(* CODESYS project HFX_research_EMMS_.project

Project tree, tasks and I/O mapping:
  Device : CR1201, ifm electronic, order no. PDM360NG, version 3.3.0.2
    application Application
      libraries: Standard, * (System); VisuDialogs, * (System); CAA CiA 405, 3.5.8.0 (CAA Technical Workgroup)
      task MainTask (cyclic, interval t#20ms, priority 1) calls PLC_PRG
      task VISU_TASK (cyclic, interval t#20ms, priority 15) calls VisuElems.Visu_Prg
      task TrendRecordingTask (cyclic, interval 100 ms, priority 31) calls VisuTrendStorageAccess.GlobalInstances.g_TrendRecordingManager.CyclicCall
      program PLC_PRG [ST]
      visualisation Main_sys
      visualisation Battery_sys
      visualisation Hydrogen_Fuel_cell_sys
      visualisation Main_Overview
      visualisation Hydrogen_Tanks
      visualisation Machine_system_properties
      visualisation Control_System_Simulation
      visualisation Visualization
      visualisation electric_motor
      visualisation Hydraulic_System
      visualisation Cooling_system
      visualisation camera_system
      image pool ImagePool
    System_Info : System_Info, ifm electronic, version 3.3.0.2
    Local_IO : Local IO, ifm electronic, version 3.3.0.2
      Inputs : Inputs, ifm electronic, version 3.3.0.2
          input  IN0000 : IN_MULTIFUNCTION_B_INPUT_MAPPING_TYPE  // IN0000
      Outputs : Outputs, ifm electronic, version 3.3.0.2
          output OUT0000 : OUT_DIGITAL_A_OUTPUT_MAPPING_TYPE  // OUT0000
      System_Inputs : System_Inputs, ifm electronic, version 3.3.0.2
          input  uiVoltageVBB30 : UINT  // Voltage VBB30
          input  uiVoltageVBB15 : UINT  // Voltage VBB15
          input  iTemperature0 : INT  // Board Temperature 0
          input  iTemperature1 : INT  // Board Temperature 1
          input  uiLightSensor : UINT  // Light Sensor
    HMI : HMI, ifm electronic, version 3.3.0.2
      User_LEDs : User_LEDs, ifm electronic, version 3.3.0.2
          output LED0 : LED_IEC_A_OUTPUT_MAPPING_TYPE  // User LED 0
      LCD_Backlight : LCD Backlight, ifm electronic, version 3.3.0.2
          output uiBacklightBrightness AT %QW5 : UINT  // Brightness
      Buzzer : Buzzer, ifm electronic, version 3.3.0.2
          output uiBuzzerFreq : UINT  // Frequency
          output xBuzzerON : BIT  // Buzzer ON
      KeyBoards : KeyBoards, ifm electronic, version 3.3.0.2
        Key_Backlight_settings : Key Backlight settings, ifm electronic, version 3.3.0.2
            output xNightModeON AT %QX14.1 : BIT  // Night Mode ON
        Key_Mapping : Key Mapping, ifm electronic, version 3.3.0.2
        Keys : Keys, ifm electronic, version 3.3.0.2
          LEDs_Keyboard_1 : LEDs Keyboard 1, ifm electronic, version 3.3.0.2
              output LEDsKeyboard1 AT %QW8 : WORD  // LEDsKeyboard1
          LEDs_Keyboard_3 : LEDs Keyboard 3, ifm electronic, version 3.3.0.2
              output LEDsKeyboard3 AT %QW9 : WORD  // LEDs Keyboard 3
    Communication : Communication, ifm electronic, version 3.3.0.2
      Ethernet : Ethernet, ifm electronic, version 3.3.0.2
      CAN : CAN, ifm electronic, version 3.3.0.2
        CANbus : CANbus, ifm electronic, version 1.0.0.0
            settings: Baudrate = 125; NetID = 1
          CANopen_Manager : CANopen_Manager, 3S - Smart Software Solutions GmbH, version 3.5.7.20
              settings: ConfigVersion = 50659584
            JN2100 : JN2100, ifm electornic GmbH, order no. JN2100, version Revision=16#000000AA, FileVersion=1.1, File=inclinationsensor_JNJN2100_V2.5.4.eds
                settings: General Options.Create all SDOs = TRUE; NODEIDSAVED = 10; SDO Timeout = 1000000; Explicit Deactivate PDOs = TRUE; PDO_Autoconfig = FALSE; EXPERTSETTINGS = True; Emergency-General Parameters.Emergency COBID = 16#0000008A; Heartbeat-Producer Time = 200; PDO 16#1800.COBID = 16#0000018A; PDO 16#1800.Transmission Type = 16#FE; Process by CANopenManager = TRUE; PDO 16#1801.COBID = 16#0000028A; PDO 16#1801.Transmission Type = 16#FE; Process by CANopenManager = TRUE; PDO 16#1802.COBID = 16#0000038A; PDO 16#1802.Transmission Type = 16#FE; Process by CANopenManager = TRUE; PDO 16#1803.COBID = 16#0000048A; PDO 16#1803.Transmission Type = 16#FE; Process by CANopenManager = TRUE; Slope long16.Subindex = 16#00; Slope lateral16.Subindex = 16#00; Slope long32.Subindex = 16#00; Slope lateral32.Subindex = 16#00; v effektive vector magnitude.Subindex = 16#00; a peak vector magnitude.Subindex = 16#00; a x vector.Subindex = 16#00; a y vector.Subindex = 16#00; a z vector.Subindex = 16#00; SDO List.Set Guardtime.Index = 16#100C; SDO List.Set Guardtime.Subindex = 16#00; SDO List.Set Guardtime.Value = 16#00000000; SDO List.Set Guardtime.Size = 16; SDO List.Set Guardtime.AbortIfError = FALSE; SDO List.Set Guardtime.JumpToLine = FALSE; SDO List.Set Guardtime.Line = 0; SDO List.Set Lifetime.Index = 16#100D; SDO List.Set Lifetime.Subindex = 16#00; SDO List.Set Lifetime.Value = 16#00000000; SDO List.Set Lifetime.Size = 8;
                  SDO List.Set Lifetime.AbortIfError = FALSE; SDO List.Set Lifetime.JumpToLine = FALSE; SDO List.Set Lifetime.Line = 0; SDO List.Set Heartbeat Producer.Index = 16#1017; SDO List.Set Heartbeat Producer.Subindex = 16#00; SDO List.Set Heartbeat Producer.Value = 16#000000C8; SDO List.Set Heartbeat Producer.Size = 16; SDO List.Set Heartbeat Producer.AbortIfError = FALSE; SDO List.Set Heartbeat Producer.JumpToLine = FALSE; SDO List.Set Heartbeat Producer.Line = 0; SDO List.Disable PDO.Index = 16#1800; SDO List.Disable PDO.Subindex = 16#01; SDO List.Disable PDO.Value = 16#8000018A; SDO List.Disable PDO.Size = 32; SDO List.Disable PDO.AbortIfError = FALSE; SDO List.Disable PDO.JumpToLine = FALSE; SDO List.Disable PDO.Line = 0; SDO List.Set transmission type.Index = 16#1800; SDO List.Set transmission type.Subindex = 16#02; SDO List.Set transmission type.Value = 16#FE; SDO List.Set transmission type.Size = 8; SDO List.Set transmission type.AbortIfError = FALSE; SDO List.Set transmission type.JumpToLine = FALSE; SDO List.Set transmission type.Line = 0; SDO List.Set inhibit time.Index = 16#1800; SDO List.Set inhibit time.Subindex = 16#03; SDO List.Set inhibit time.Value = 16#0000; SDO List.Set inhibit time.Size = 16; SDO List.Set inhibit time.AbortIfError = FALSE; SDO List.Set inhibit time.JumpToLine = FALSE; SDO List.Set inhibit time.Line = 0; SDO List.Set event time.Index = 16#1800; SDO List.Set event time.Subindex = 16#05; SDO List.Set event time.Value = 16#000A; SDO List.Set event time.Size = 16; SDO List.Set event time.AbortIfError = FALSE; SDO List.Set event time.JumpToLine = FALSE; SDO List.Set event time.Line = 0; SDO List.Clear pdo mapping.Index = 16#1A00; SDO List.Clear pdo mapping.Subindex = 16#00;
                  SDO List.Clear pdo mapping.Value = 16#0; SDO List.Clear pdo mapping.Size = 8; SDO List.Clear pdo mapping.AbortIfError = FALSE; SDO List.Clear pdo mapping.JumpToLine = FALSE; SDO List.Clear pdo mapping.Line = 0; SDO List.Set Mapping.Index = 16#1A00; SDO List.Set Mapping.Subindex = 16#01; SDO List.Set Mapping.Value = 16#60100010; SDO List.Set Mapping.Size = 32; SDO List.Set Mapping.AbortIfError = FALSE; SDO List.Set Mapping.JumpToLine = FALSE; SDO List.Set Mapping.Line = 0; SDO List.Set Mapping.Index = 16#1A00; SDO List.Set Mapping.Subindex = 16#02; SDO List.Set Mapping.Value = 16#60200010; SDO List.Set Mapping.Size = 32; SDO List.Set Mapping.AbortIfError = FALSE; SDO List.Set Mapping.JumpToLine = FALSE; SDO List.Set Mapping.Line = 0; SDO List.Set number of mappings.Index = 16#1A00; SDO List.Set number of mappings.Subindex = 16#00; SDO List.Set number of mappings.Value = 16#02; SDO List.Set number of mappings.Size = 8; SDO List.Set number of mappings.AbortIfError = FALSE; SDO List.Set number of mappings.JumpToLine = FALSE; SDO List.Set number of mappings.Line = 0; SDO List.Set and enable COB-ID.Index = 16#1800; SDO List.Set and enable COB-ID.Subindex = 16#01; SDO List.Set and enable COB-ID.Value = 16#0000018A; SDO List.Set and enable COB-ID.Size = 32; SDO List.Set and enable COB-ID.AbortIfError = FALSE; SDO List.Set and enable COB-ID.JumpToLine = FALSE; SDO List.Set and enable COB-ID.Line = 0; SDO List.Disable PDO.Index = 16#1801; SDO List.Disable PDO.Subindex = 16#01; SDO List.Disable PDO.Value = 16#8000028A; SDO List.Disable PDO.Size = 32; SDO List.Disable PDO.AbortIfError = FALSE; SDO List.Disable PDO.JumpToLine = FALSE; SDO List.Disable PDO.Line = 0;
                  SDO List.Set transmission type.Index = 16#1801; SDO List.Set transmission type.Subindex = 16#02; SDO List.Set transmission type.Value = 16#FE; SDO List.Set transmission type.Size = 8; SDO List.Set transmission type.AbortIfError = FALSE; SDO List.Set transmission type.JumpToLine = FALSE; SDO List.Set transmission type.Line = 0; SDO List.Set inhibit time.Index = 16#1801; SDO List.Set inhibit time.Subindex = 16#03; SDO List.Set inhibit time.Value = 16#0000; SDO List.Set inhibit time.Size = 16; SDO List.Set inhibit time.AbortIfError = FALSE; SDO List.Set inhibit time.JumpToLine = FALSE; SDO List.Set inhibit time.Line = 0; SDO List.Set event time.Index = 16#1801; SDO List.Set event time.Subindex = 16#05; SDO List.Set event time.Value = 16#000A; SDO List.Set event time.Size = 16; SDO List.Set event time.AbortIfError = FALSE; SDO List.Set event time.JumpToLine = FALSE; SDO List.Set event time.Line = 0; SDO List.Clear pdo mapping.Index = 16#1A01; SDO List.Clear pdo mapping.Subindex = 16#00; SDO List.Clear pdo mapping.Value = 16#0; SDO List.Clear pdo mapping.Size = 8; SDO List.Clear pdo mapping.AbortIfError = FALSE; SDO List.Clear pdo mapping.JumpToLine = FALSE; SDO List.Clear pdo mapping.Line = 0; SDO List.Set Mapping.Index = 16#1A01; SDO List.Set Mapping.Subindex = 16#01; SDO List.Set Mapping.Value = 16#61100020; SDO List.Set Mapping.Size = 32; SDO List.Set Mapping.AbortIfError = FALSE; SDO List.Set Mapping.JumpToLine = FALSE; SDO List.Set Mapping.Line = 0; SDO List.Set Mapping.Index = 16#1A01; SDO List.Set Mapping.Subindex = 16#02; SDO List.Set Mapping.Value = 16#61200020; SDO List.Set Mapping.Size = 32; SDO List.Set Mapping.AbortIfError = FALSE;
                  SDO List.Set Mapping.JumpToLine = FALSE; SDO List.Set Mapping.Line = 0; SDO List.Set number of mappings.Index = 16#1A01; SDO List.Set number of mappings.Subindex = 16#00; SDO List.Set number of mappings.Value = 16#02; SDO List.Set number of mappings.Size = 8; SDO List.Set number of mappings.AbortIfError = FALSE; SDO List.Set number of mappings.JumpToLine = FALSE; SDO List.Set number of mappings.Line = 0; SDO List.Set and enable COB-ID.Index = 16#1801; SDO List.Set and enable COB-ID.Subindex = 16#01; SDO List.Set and enable COB-ID.Value = 16#0000028A; SDO List.Set and enable COB-ID.Size = 32; SDO List.Set and enable COB-ID.AbortIfError = FALSE; SDO List.Set and enable COB-ID.JumpToLine = FALSE; SDO List.Set and enable COB-ID.Line = 0; SDO List.Disable PDO.Index = 16#1802; SDO List.Disable PDO.Subindex = 16#01; SDO List.Disable PDO.Value = 16#8000038A; SDO List.Disable PDO.Size = 32; SDO List.Disable PDO.AbortIfError = FALSE; SDO List.Disable PDO.JumpToLine = FALSE; SDO List.Disable PDO.Line = 0; SDO List.Set transmission type.Index = 16#1802; SDO List.Set transmission type.Subindex = 16#02; SDO List.Set transmission type.Value = 16#FE; SDO List.Set transmission type.Size = 8; SDO List.Set transmission type.AbortIfError = FALSE; SDO List.Set transmission type.JumpToLine = FALSE; SDO List.Set transmission type.Line = 0; SDO List.Set inhibit time.Index = 16#1802; SDO List.Set inhibit time.Subindex = 16#03; SDO List.Set inhibit time.Value = 16#0000; SDO List.Set inhibit time.Size = 16; SDO List.Set inhibit time.AbortIfError = FALSE; SDO List.Set inhibit time.JumpToLine = FALSE; SDO List.Set inhibit time.Line = 0; SDO List.Set event time.Index = 16#1802; SDO List.Set event time.Subindex = 16#05; SDO List.Set event time.Value = 16#000A;
                  SDO List.Set event time.Size = 16; SDO List.Set event time.AbortIfError = FALSE; SDO List.Set event time.JumpToLine = FALSE; SDO List.Set event time.Line = 0; SDO List.Clear pdo mapping.Index = 16#1A02; SDO List.Clear pdo mapping.Subindex = 16#00; SDO List.Clear pdo mapping.Value = 16#0; SDO List.Clear pdo mapping.Size = 8; SDO List.Clear pdo mapping.AbortIfError = FALSE; SDO List.Clear pdo mapping.JumpToLine = FALSE; SDO List.Clear pdo mapping.Line = 0; SDO List.Set Mapping.Index = 16#1A02; SDO List.Set Mapping.Subindex = 16#01; SDO List.Set Mapping.Value = 16#5C100020; SDO List.Set Mapping.Size = 32; SDO List.Set Mapping.AbortIfError = FALSE; SDO List.Set Mapping.JumpToLine = FALSE; SDO List.Set Mapping.Line = 0; SDO List.Set Mapping.Index = 16#1A02; SDO List.Set Mapping.Subindex = 16#02; SDO List.Set Mapping.Value = 16#5C110020; SDO List.Set Mapping.Size = 32; SDO List.Set Mapping.AbortIfError = FALSE; SDO List.Set Mapping.JumpToLine = FALSE; SDO List.Set Mapping.Line = 0; SDO List.Set number of mappings.Index = 16#1A02; SDO List.Set number of mappings.Subindex = 16#00; SDO List.Set number of mappings.Value = 16#02; SDO List.Set number of mappings.Size = 8; SDO List.Set number of mappings.AbortIfError = FALSE; SDO List.Set number of mappings.JumpToLine = FALSE; SDO List.Set number of mappings.Line = 0; SDO List.Set and enable COB-ID.Index = 16#1802; SDO List.Set and enable COB-ID.Subindex = 16#01; SDO List.Set and enable COB-ID.Value = 16#0000038A; SDO List.Set and enable COB-ID.Size = 32; SDO List.Set and enable COB-ID.AbortIfError = FALSE; SDO List.Set and enable COB-ID.JumpToLine = FALSE; SDO List.Set and enable COB-ID.Line = 0; SDO List.Disable PDO.Index = 16#1803;
                  SDO List.Disable PDO.Subindex = 16#01; SDO List.Disable PDO.Value = 16#8000048A; SDO List.Disable PDO.Size = 32; SDO List.Disable PDO.AbortIfError = FALSE; SDO List.Disable PDO.JumpToLine = FALSE; SDO List.Disable PDO.Line = 0; SDO List.Set transmission type.Index = 16#1803; SDO List.Set transmission type.Subindex = 16#02; SDO List.Set transmission type.Value = 16#FE; SDO List.Set transmission type.Size = 8; SDO List.Set transmission type.AbortIfError = FALSE; SDO List.Set transmission type.JumpToLine = FALSE; SDO List.Set transmission type.Line = 0; SDO List.Set inhibit time.Index = 16#1803; SDO List.Set inhibit time.Subindex = 16#03; SDO List.Set inhibit time.Value = 16#0000; SDO List.Set inhibit time.Size = 16; SDO List.Set inhibit time.AbortIfError = FALSE; SDO List.Set inhibit time.JumpToLine = FALSE; SDO List.Set inhibit time.Line = 0; SDO List.Set event time.Index = 16#1803; SDO List.Set event time.Subindex = 16#05; SDO List.Set event time.Value = 16#000A; SDO List.Set event time.Size = 16; SDO List.Set event time.AbortIfError = FALSE; SDO List.Set event time.JumpToLine = FALSE; SDO List.Set event time.Line = 0; SDO List.Clear pdo mapping.Index = 16#1A03; SDO List.Clear pdo mapping.Subindex = 16#00; SDO List.Clear pdo mapping.Value = 16#0; SDO List.Clear pdo mapping.Size = 8; SDO List.Clear pdo mapping.AbortIfError = FALSE; SDO List.Clear pdo mapping.JumpToLine = FALSE; SDO List.Clear pdo mapping.Line = 0; SDO List.Set Mapping.Index = 16#1A03; SDO List.Set Mapping.Subindex = 16#01; SDO List.Set Mapping.Value = 16#5D100010; SDO List.Set Mapping.Size = 32; SDO List.Set Mapping.AbortIfError = FALSE; SDO List.Set Mapping.JumpToLine = FALSE;
                  SDO List.Set Mapping.Line = 0; SDO List.Set Mapping.Index = 16#1A03; SDO List.Set Mapping.Subindex = 16#02; SDO List.Set Mapping.Value = 16#5D110010; SDO List.Set Mapping.Size = 32; SDO List.Set Mapping.AbortIfError = FALSE; SDO List.Set Mapping.JumpToLine = FALSE; SDO List.Set Mapping.Line = 0; SDO List.Set Mapping.Index = 16#1A03; SDO List.Set Mapping.Subindex = 16#03; SDO List.Set Mapping.Value = 16#5D120010; SDO List.Set Mapping.Size = 32; SDO List.Set Mapping.AbortIfError = FALSE; SDO List.Set Mapping.JumpToLine = FALSE; SDO List.Set Mapping.Line = 0; SDO List.Set number of mappings.Index = 16#1A03; SDO List.Set number of mappings.Subindex = 16#00; SDO List.Set number of mappings.Value = 16#03; SDO List.Set number of mappings.Size = 8; SDO List.Set number of mappings.AbortIfError = FALSE; SDO List.Set number of mappings.JumpToLine = FALSE; SDO List.Set number of mappings.Line = 0; SDO List.Set and enable COB-ID.Index = 16#1803; SDO List.Set and enable COB-ID.Subindex = 16#01; SDO List.Set and enable COB-ID.Value = 16#0000048A; SDO List.Set and enable COB-ID.Size = 32; SDO List.Set and enable COB-ID.AbortIfError = FALSE; SDO List.Set and enable COB-ID.JumpToLine = FALSE; SDO List.Set and enable COB-ID.Line = 0; SDO List.Node ID.Index = 16#2000; SDO List.Node ID.Subindex = 16#00; SDO List.Node ID.Value = 10; SDO List.Node ID.Size = 8; SDO List.Node ID.AbortIfError = FALSE; SDO List.Node ID.JumpToLine = FALSE; SDO List.Node ID.Line = 0; SDO List.Baudrate [kbit].Index = 16#2001; SDO List.Baudrate [kbit].Subindex = 16#00; SDO List.Baudrate [kbit].Value = 125; SDO List.Baudrate [kbit].Size = 16;
                  SDO List.Baudrate [kbit].AbortIfError = FALSE; SDO List.Baudrate [kbit].JumpToLine = FALSE; SDO List.Baudrate [kbit].Line = 0; SDO List.Microcontroller Reset.Index = 16#2002; SDO List.Microcontroller Reset.Subindex = 16#00; SDO List.Microcontroller Reset.Value = 0; SDO List.Microcontroller Reset.Size = 8; SDO List.Microcontroller Reset.AbortIfError = FALSE; SDO List.Microcontroller Reset.JumpToLine = FALSE; SDO List.Microcontroller Reset.Line = 0; SDO List.Quadrant Correction.Index = 16#2040; SDO List.Quadrant Correction.Subindex = 16#00; SDO List.Quadrant Correction.Value = 2; SDO List.Quadrant Correction.Size = 8; SDO List.Quadrant Correction.AbortIfError = FALSE; SDO List.Quadrant Correction.JumpToLine = FALSE; SDO List.Quadrant Correction.Line = 0; SDO List.Heater On.Index = 16#2041; SDO List.Heater On.Subindex = 16#00; SDO List.Heater On.Value = 1; SDO List.Heater On.Size = 8; SDO List.Heater On.AbortIfError = FALSE; SDO List.Heater On.JumpToLine = FALSE; SDO List.Heater On.Line = 0; SDO List.Teach Index.Index = 16#2042; SDO List.Teach Index.Subindex = 16#00; SDO List.Teach Index.Value = 2; SDO List.Teach Index.Size = 8; SDO List.Teach Index.AbortIfError = FALSE; SDO List.Teach Index.JumpToLine = FALSE; SDO List.Teach Index.Line = 0; SDO List.FIR Filter Angle.Index = 16#2043; SDO List.FIR Filter Angle.Subindex = 16#00; SDO List.FIR Filter Angle.Value = 2; SDO List.FIR Filter Angle.Size = 8; SDO List.FIR Filter Angle.AbortIfError = FALSE; SDO List.FIR Filter Angle.JumpToLine = FALSE; SDO List.FIR Filter Angle.Line = 0; SDO List.Angle Calculation Algorithm.Index = 16#2044; SDO List.Angle Calculation Algorithm.Subindex = 16#00;
                  SDO List.Angle Calculation Algorithm.Value = 0; SDO List.Angle Calculation Algorithm.Size = 8; SDO List.Angle Calculation Algorithm.AbortIfError = FALSE; SDO List.Angle Calculation Algorithm.JumpToLine = FALSE; SDO List.Angle Calculation Algorithm.Line = 0; SDO List.CAN 120 Ohm Resistor.Index = 16#2045; SDO List.CAN 120 Ohm Resistor.Subindex = 16#00; SDO List.CAN 120 Ohm Resistor.Value = 1; SDO List.CAN 120 Ohm Resistor.Size = 8; SDO List.CAN 120 Ohm Resistor.AbortIfError = FALSE; SDO List.CAN 120 Ohm Resistor.JumpToLine = FALSE; SDO List.CAN 120 Ohm Resistor.Line = 0; SDO List.Zero Index.Index = 16#2046; SDO List.Zero Index.Subindex = 16#00; SDO List.Zero Index.Value = 2; SDO List.Zero Index.Size = 8; SDO List.Zero Index.AbortIfError = FALSE; SDO List.Zero Index.JumpToLine = FALSE; SDO List.Zero Index.Line = 0; SDO List.Measurement Output.Index = 16#2047; SDO List.Measurement Output.Subindex = 16#00; SDO List.Measurement Output.Value = 0; SDO List.Measurement Output.Size = 8; SDO List.Measurement Output.AbortIfError = FALSE; SDO List.Measurement Output.JumpToLine = FALSE; SDO List.Measurement Output.Line = 0; SDO List.Axis Selection v eff - a peak.Index = 16#2048; SDO List.Axis Selection v eff - a peak.Subindex = 16#00; SDO List.Axis Selection v eff - a peak.Value = 7; SDO List.Axis Selection v eff - a peak.Size = 8; SDO List.Axis Selection v eff - a peak.AbortIfError = FALSE; SDO List.Axis Selection v eff - a peak.JumpToLine = FALSE; SDO List.Axis Selection v eff - a peak.Line = 0; SDO List.FIR Filter v eff - a peak.Index = 16#2049; SDO List.FIR Filter v eff - a peak.Subindex = 16#00; SDO List.FIR Filter v eff - a peak.Value = 5; SDO List.FIR Filter v eff - a peak.Size = 8; SDO List.FIR Filter v eff - a peak.AbortIfError = FALSE; SDO List.FIR Filter v eff - a peak.JumpToLine = FALSE; SDO List.FIR Filter v eff - a peak.Line = 0;
                  SDO List.Measurement Range v eff - a peak.Index = 16#204A; SDO List.Measurement Range v eff - a peak.Subindex = 16#00; SDO List.Measurement Range v eff - a peak.Value = 2; SDO List.Measurement Range v eff - a peak.Size = 8; SDO List.Measurement Range v eff - a peak.AbortIfError = FALSE; SDO List.Measurement Range v eff - a peak.JumpToLine = FALSE; SDO List.Measurement Range v eff - a peak.Line = 0; SDO List.Factory Reset.Index = 16#207F; SDO List.Factory Reset.Subindex = 16#00; SDO List.Factory Reset.Value = 0; SDO List.Factory Reset.Size = 8; SDO List.Factory Reset.AbortIfError = FALSE; SDO List.Factory Reset.JumpToLine = FALSE; SDO List.Factory Reset.Line = 0; SDO List.Activate Self Test.Index = 16#4004; SDO List.Activate Self Test.Subindex = 16#01; SDO List.Activate Self Test.Value = 0; SDO List.Activate Self Test.Size = 8; SDO List.Activate Self Test.AbortIfError = FALSE; SDO List.Activate Self Test.JumpToLine = FALSE; SDO List.Activate Self Test.Line = 0; SDO List.Resolution.Index = 16#6000; SDO List.Resolution.Subindex = 16#00; SDO List.Resolution.Value = 100; SDO List.Resolution.Size = 16; SDO List.Resolution.AbortIfError = FALSE; SDO List.Resolution.JumpToLine = FALSE; SDO List.Resolution.Line = 0; SDO List.Slope long16 operating parameter.Index = 16#6011; SDO List.Slope long16 operating parameter.Subindex = 16#00; SDO List.Slope long16 operating parameter.Value = 16#0; SDO List.Slope long16 operating parameter.Size = 8; SDO List.Slope long16 operating parameter.AbortIfError = FALSE; SDO List.Slope long16 operating parameter.JumpToLine = FALSE; SDO List.Slope long16 operating parameter.Line = 0; SDO List.Slope lateral16 operating parameter.Index = 16#6021; SDO List.Slope lateral16 operating parameter.Subindex = 16#00; SDO List.Slope lateral16 operating parameter.Value = 16#0; SDO List.Slope lateral16 operating parameter.Size = 8; SDO List.Slope lateral16 operating parameter.AbortIfError = FALSE;
                  SDO List.Slope lateral16 operating parameter.JumpToLine = FALSE; SDO List.Slope lateral16 operating parameter.Line = 0; SDO List.Slope long32 operating parameter.Index = 16#6111; SDO List.Slope long32 operating parameter.Subindex = 16#00; SDO List.Slope long32 operating parameter.Value = 16#0; SDO List.Slope long32 operating parameter.Size = 8; SDO List.Slope long32 operating parameter.AbortIfError = FALSE; SDO List.Slope long32 operating parameter.JumpToLine = FALSE; SDO List.Slope long32 operating parameter.Line = 0; SDO List.Slope lateral32 operating parameter.Index = 16#6121; SDO List.Slope lateral32 operating parameter.Subindex = 16#00; SDO List.Slope lateral32 operating parameter.Value = 16#0; SDO List.Slope lateral32 operating parameter.Size = 8; SDO List.Slope lateral32 operating parameter.AbortIfError = FALSE; SDO List.Slope lateral32 operating parameter.JumpToLine = FALSE; SDO List.Slope lateral32 operating parameter.Line = 0; ConfigVersion = 50659584
                input  Application.PLC_PRG.longi : INT  // Slope long16
                input  Application.PLC_PRG.slope : INT  // Slope lateral16
                input  Application.PLC_PRG.x_vector1 : INT  // a x vector
                input  Application.PLC_PRG.y_vector1 : INT  // a y vector
                input  Application.PLC_PRG.z_vector : INT  // a z vector
                unmapped channels: Slope long32, Slope lateral32, v effektive vector magnitude, a peak vector magnitude
        CANbus_1 : CANbus, ifm electronic, version 1.0.0.0
          CANopen_Manager_1 : CANopen_Manager, 3S - Smart Software Solutions GmbH, version 3.5.7.20
              settings: ConfigVersion = 50659584
            System_R360_I_O_CompactModule_CR2013 : System R360: I/O CompactModule CR2013, ifm electronic gmbh, order no. CR2013, version Revision=16#00000000, FileVersion=1.0, File=CR2013_board_eds.eds
                settings: NODEIDSAVED = 11; SDO Timeout = 1000000; PDO_Autoconfig = FALSE; EXPERTSETTINGS = FALSE; Nodeguarding.Guard Time = 200 ms; Nodeguarding.Life Time Factor = 2; Emergency-General Parameters.Emergency COBID = 16#4000008B; PDO 16#1400.COBID = 16#0000020B; PDO 16#1400.Transmission Type = 16#01; Process by CANopenManager = TRUE; PDO 16#1401.COBID = 16#0000030B; PDO 16#1401.Transmission Type = 16#01; Process by CANopenManager = TRUE; PDO 16#1800.COBID = 16#0000018B; PDO 16#1800.Inhibit Time = 0; PDO 16#1800.Event Timer = 0; Process by CANopenManager = TRUE; PDO 16#1801.COBID = 16#0000028B; PDO 16#1801.Transmission Type = 16#01; PDO 16#1801.Inhibit Time = 0; PDO 16#1801.Event Timer = 0; Process by CANopenManager = TRUE; binary outputs 1.Subindex = 16#01; analog output channel  1.Subindex = 16#01; analog output channel  2.Subindex = 16#02; analog output channel  3.Subindex = 16#03; analog output channel  4.Subindex = 16#04; binary inputs 1.Subindex = 16#01; analog input channel  1.Subindex = 16#01; analog input channel  2.Subindex = 16#02; analog input channel  3.Subindex = 16#03; analog input channel  4.Subindex = 16#04; SDO List.Set Guardtime.Index = 16#100C; SDO List.Set Guardtime.Subindex = 16#00; SDO List.Set Guardtime.Value = 16#000000C8; SDO List.Set Guardtime.Size = 16; SDO List.Set Guardtime.AbortIfError = FALSE; SDO List.Set Guardtime.JumpToLine = FALSE; SDO List.Set Guardtime.Line = 0; SDO List.Set Lifetime.Index = 16#100D;
                  SDO List.Set Lifetime.Subindex = 16#00; SDO List.Set Lifetime.Value = 16#00000002; SDO List.Set Lifetime.Size = 8; SDO List.Set Lifetime.AbortIfError = FALSE; SDO List.Set Lifetime.JumpToLine = FALSE; SDO List.Set Lifetime.Line = 0; SDO List.Disable Emcy CobID.Index = 16#1014; SDO List.Disable Emcy CobID.Subindex = 16#00; SDO List.Disable Emcy CobID.Value = 16#C000008B; SDO List.Disable Emcy CobID.Size = 32; SDO List.Disable Emcy CobID.AbortIfError = FALSE; SDO List.Disable Emcy CobID.JumpToLine = FALSE; SDO List.Disable Emcy CobID.Line = 0; SDO List.Set Emcy CobID.Index = 16#1014; SDO List.Set Emcy CobID.Subindex = 16#00; SDO List.Set Emcy CobID.Value = 16#4000008B; SDO List.Set Emcy CobID.Size = 32; SDO List.Set Emcy CobID.AbortIfError = FALSE; SDO List.Set Emcy CobID.JumpToLine = FALSE; SDO List.Set Emcy CobID.Line = 0; SDO List.Disable PDO.Index = 16#1400; SDO List.Disable PDO.Subindex = 16#01; SDO List.Disable PDO.Value = 16#8000020B; SDO List.Disable PDO.Size = 32; SDO List.Disable PDO.AbortIfError = FALSE; SDO List.Disable PDO.JumpToLine = FALSE; SDO List.Disable PDO.Line = 0; SDO List.Set transmission type.Index = 16#1400; SDO List.Set transmission type.Subindex = 16#02; SDO List.Set transmission type.Value = 16#01; SDO List.Set transmission type.Size = 8; SDO List.Set transmission type.AbortIfError = FALSE; SDO List.Set transmission type.JumpToLine = FALSE; SDO List.Set transmission type.Line = 0; SDO List.Set and enable COB-ID.Index = 16#1400; SDO List.Set and enable COB-ID.Subindex = 16#01; SDO List.Set and enable COB-ID.Value = 16#0000020B; SDO List.Set and enable COB-ID.Size = 32; SDO List.Set and enable COB-ID.AbortIfError = FALSE; SDO List.Set and enable COB-ID.JumpToLine = FALSE;
                  SDO List.Set and enable COB-ID.Line = 0; SDO List.Disable PDO.Index = 16#1401; SDO List.Disable PDO.Subindex = 16#01; SDO List.Disable PDO.Value = 16#8000030B; SDO List.Disable PDO.Size = 32; SDO List.Disable PDO.AbortIfError = FALSE; SDO List.Disable PDO.JumpToLine = FALSE; SDO List.Disable PDO.Line = 0; SDO List.Set transmission type.Index = 16#1401; SDO List.Set transmission type.Subindex = 16#02; SDO List.Set transmission type.Value = 16#01; SDO List.Set transmission type.Size = 8; SDO List.Set transmission type.AbortIfError = FALSE; SDO List.Set transmission type.JumpToLine = FALSE; SDO List.Set transmission type.Line = 0; SDO List.Set and enable COB-ID.Index = 16#1401; SDO List.Set and enable COB-ID.Subindex = 16#01; SDO List.Set and enable COB-ID.Value = 16#0000030B; SDO List.Set and enable COB-ID.Size = 32; SDO List.Set and enable COB-ID.AbortIfError = FALSE; SDO List.Set and enable COB-ID.JumpToLine = FALSE; SDO List.Set and enable COB-ID.Line = 0; SDO List.Disable PDO.Index = 16#1800; SDO List.Disable PDO.Subindex = 16#01; SDO List.Disable PDO.Value = 16#8000018B; SDO List.Disable PDO.Size = 32; SDO List.Disable PDO.AbortIfError = FALSE; SDO List.Disable PDO.JumpToLine = FALSE; SDO List.Disable PDO.Line = 0; SDO List.Set transmission type.Index = 16#1800; SDO List.Set transmission type.Subindex = 16#02; SDO List.Set transmission type.Value = 16#FF; SDO List.Set transmission type.Size = 8; SDO List.Set transmission type.AbortIfError = FALSE; SDO List.Set transmission type.JumpToLine = FALSE; SDO List.Set transmission type.Line = 0; SDO List.Set and enable COB-ID.Index = 16#1800; SDO List.Set and enable COB-ID.Subindex = 16#01; SDO List.Set and enable COB-ID.Value = 16#0000018B; SDO List.Set and enable COB-ID.Size = 32;
                  SDO List.Set and enable COB-ID.AbortIfError = FALSE; SDO List.Set and enable COB-ID.JumpToLine = FALSE; SDO List.Set and enable COB-ID.Line = 0; SDO List.Disable PDO.Index = 16#1801; SDO List.Disable PDO.Subindex = 16#01; SDO List.Disable PDO.Value = 16#8000028B; SDO List.Disable PDO.Size = 32; SDO List.Disable PDO.AbortIfError = FALSE; SDO List.Disable PDO.JumpToLine = FALSE; SDO List.Disable PDO.Line = 0; SDO List.Set transmission type.Index = 16#1801; SDO List.Set transmission type.Subindex = 16#02; SDO List.Set transmission type.Value = 16#01; SDO List.Set transmission type.Size = 8; SDO List.Set transmission type.AbortIfError = FALSE; SDO List.Set transmission type.JumpToLine = FALSE; SDO List.Set transmission type.Line = 0; SDO List.Set and enable COB-ID.Index = 16#1801; SDO List.Set and enable COB-ID.Subindex = 16#01; SDO List.Set and enable COB-ID.Value = 16#0000028B; SDO List.Set and enable COB-ID.Size = 32; SDO List.Set and enable COB-ID.AbortIfError = FALSE; SDO List.Set and enable COB-ID.JumpToLine = FALSE; SDO List.Set and enable COB-ID.Line = 0; ConfigVersion = 50659584
                unmapped channels: binary outputs 1, analog output channel  1, analog output channel  2, analog output channel  3, analog output channel  4, binary inputs 1, analog input channel  1, analog input channel  2, analog input channel  3, analog input channel  4
  libraries: VisuSymbols, 3.5.8.0 (System)
  text list GlobalTextList
  text list System
  5ce3da45-db07-42e7-a21c-a00fff4ed8f6|C:\Users\Tailly\Desktop\Picture1.png
  5ce3da45-db07-42e7-a21c-a00fff4ed8f6|C:\Users\Tailly\Desktop\CODESYS_SOFTWARE\Icons\temperature_icons.png
  5ce3da45-db07-42e7-a21c-a00fff4ed8f6|C:\Users\HFX Internship\Documents\HFX Documents and Files\3D Models\Model module e-excavator\Solidworks Models\battery only.png
  5ce3da45-db07-42e7-a21c-a00fff4ed8f6|C:\Users\HFX Internship\Documents\HFX Documents and Files\3D Models\Model module e-excavator\Solidworks Models\tank only.png
*)

// Device/Application/PLC_PRG
PROGRAM PLC_PRG
VAR
	// Hydrogen Tanks
	tank1:REAL; charge1: BOOL; rate1: INT; vrate1: INT;
	tank12:REAL; charge12: BOOL; rate12: INT; vrate12: INT;
	tank13:REAL; charge13: BOOL; rate13: INT; vrate13: INT;
	tanktot:REAL; chargetot: BOOL; ratetot: INT; vratetot: INT;
	
	// e-motor capacity
	tank2:REAL; charge2: BOOL; rate2: INT; vrate2: INT;
	// Hydrogen fuel cell
	tank3:REAL; charge3: BOOL; rate3: INT; vrate3: INT;
	// Battery equivalent energy
	tank4:REAL; charge4: BOOL; rate4: INT; vrate4: INT;
	// Hydraulic system
	tank5:REAL; charge5: BOOL; rate5: INT; vrate5: INT;
	// cooling system in general
	tank6:REAL; charge6: BOOL; rate6: INT; vrate6: INT;
	// keyboard on

	// inclination sensor variables
	slope: INT:=0; longi:INT ; x_vector1: INT := 0; y_vector1: INT:= 0; z_vector: INT;
END_VAR

 

//Hydrogen Tanks
//Tank 1
IF tank1<100 THEN
	charge1:=FALSE;
	tank1:=tank1+0.1*rate1/100;
END_IF
IF tank1>=0 THEN
	tank1:=tank1-0.1*vrate1/100;
END_IF
IF tank1>=100 THEN
	tank1:=100;
	charge1:=TRUE;
END_IF

//tank 2
IF tank12<100 THEN
	charge12:=FALSE;
	tank12:=tank12+0.1*rate12/100;
END_IF
IF tank12>=0 THEN
	tank12:=tank12-0.1*vrate12/100;
END_IF
IF tank12>=100 THEN
	tank12:=100;
	charge12:=TRUE;
END_IF

//tank3

//total tanks (1+2+3)


// emotor capacity
IF tank2<145 THEN
	charge2:=FALSE;
	tank2:=tank2+0.1*rate2/145;
END_IF
IF tank2>=0 THEN
	tank2:=tank2-0.1*vrate2/145;
END_IF
IF tank2>=145 THEN
	tank2:=145;
	charge2:=TRUE;
END_IF

// Hydrogen Fuel cell
IF tank3<100 THEN
	charge3:=FALSE;
	tank3:=tank3+0.1*rate3/100;
END_IF
IF tank3>=0 THEN
	tank3:=tank3-0.1*vrate3/100;
END_IF
IF tank3>=100 THEN
	tank3:=100;
	charge3:=TRUE;
END_IF

// Battery equivalent energy
IF tank4<100 THEN
	charge4:=FALSE;
	tank4:=tank4+0.1*rate4/100;
END_IF
IF tank4>=0 THEN
	tank4:=tank4-0.1*vrate4/100;
END_IF
IF tank4>=100 THEN
	tank4:=100;
	charge4:=TRUE;
END_IF

// Hydraulic system
IF tank5<100 THEN
	charge5:=FALSE;
	tank5:=tank5+0.1*rate5/100;
END_IF
IF tank5>=0 THEN
	tank5:=tank5-0.1*vrate5/100;
END_IF
IF tank5>=100 THEN
	tank5:=100;
	charge5:=TRUE;
END_IF

//cooling system
IF tank6<100 THEN
	charge6:=FALSE;
	tank6:=tank6+0.1*rate6/100;
END_IF
IF tank6>=0 THEN
	tank6:=tank6-0.1*vrate6/100;
END_IF
IF tank6>=100 THEN
	tank6:=100;
	charge6:=TRUE;
END_IF

IF longi >= 0 THEN
	charge1:= TRUE;
END_IF
IF slope >= 0 THEN
	charge1:= TRUE;
END_IF

END_PROGRAM

// Device/Application/Main_sys
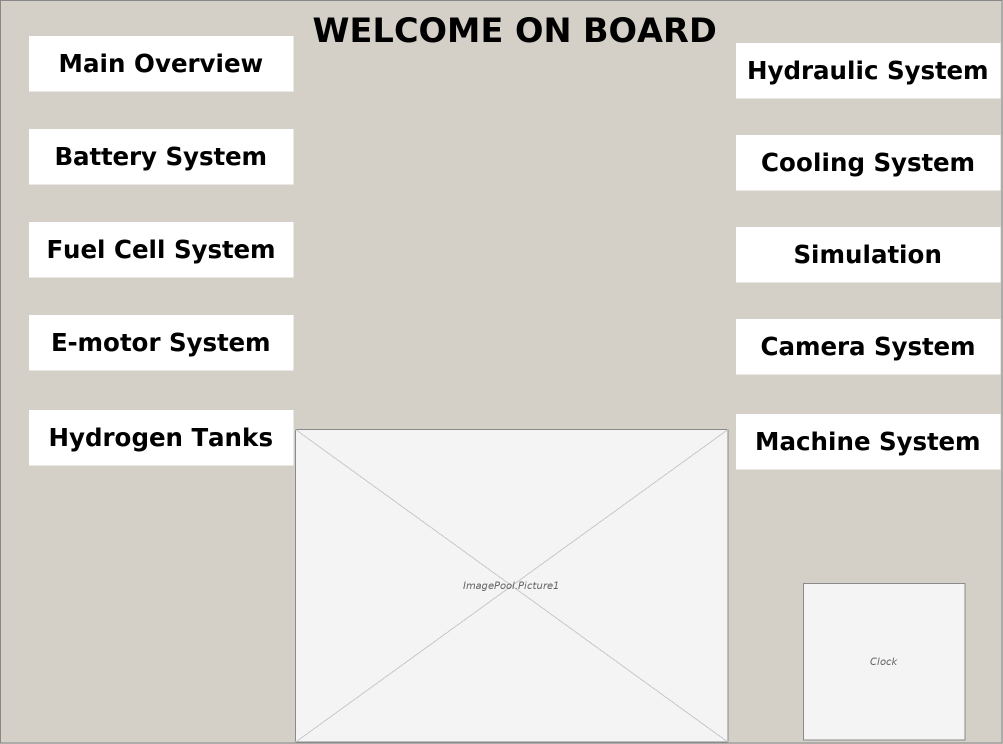
VISUALIZATION Main_sys  // 1003x744
    Group (28,35 266x431)
        Textfield (0,0 266x57), "Main Overview"
            OnMouseClick:  Assign=Main_Overview, Type=Assignment
            OnMouseClick: execute {
                IF %QX17.0 := TRUE THEN
                	%QX17.1 := FALSE;
                	%QX17.0:= TRUE;
                	%QX17.2:= FALSE;
                	%QX17.3:= FALSE;
                	%QX17.5:= FALSE;
                	%QX17.4:= FALSE;
                	%QX17.6:= FALSE;
                	%QX17.7:= FALSE;
                END_IF
            }
        Textfield (0,93 266x57), "Battery System"
            OnMouseClick:  Assign=Battery_sys, Type=Assignment
            OnMouseClick: execute {
                IF %QX17.1 := TRUE THEN
                	%QX17.1 := TRUE;
                	%QX17.0:= FALSE;
                	%QX17.2:= FALSE;
                	%QX17.3:= FALSE;
                	%QX17.5:= FALSE;
                	%QX17.4:= FALSE;
                	%QX17.6:= FALSE;
                	%QX17.7:= FALSE;
                END_IF
            }
        Textfield (0,186 266x57), "Fuel Cell System"
            OnMouseClick:  Assign=Hydrogen_Fuel_cell_sys, Type=Assignment
            OnMouseClick: execute {
                IF %QX17.2 := TRUE THEN
                	%QX17.1 := FALSE;
                	%QX17.0:= FALSE;
                	%QX17.2:= TRUE;
                	%QX17.3:= FALSE;
                	%QX17.5:= FALSE;
                	%QX17.4:= FALSE;
                	%QX17.6:= FALSE;
                	%QX17.7:= FALSE;
                END_IF
            }
        Textfield (0,279 266x57), "E-motor System"
            OnMouseClick:  Assign=electric_motor, Type=Assignment
            OnMouseClick: execute {
                IF %QX17.3 := TRUE THEN
                	%QX17.1 := FALSE;
                	%QX17.0:= FALSE;
                	%QX17.2:= FALSE;
                	%QX17.3:= TRUE;
                	%QX17.5:= FALSE;
                	%QX17.4:= FALSE;
                	%QX17.6:= FALSE;
                	%QX17.7:= FALSE;
                END_IF
            }
        Textfield (0,374 266x57), "Hydrogen Tanks"
            OnMouseClick:  Assign=Hydrogen_Tanks, Type=Assignment
            OnMouseClick: execute {
                IF %QX17.4 := TRUE THEN
                	%QX17.1 := FALSE;
                	%QX17.0:= FALSE;
                	%QX17.2:= FALSE;
                	%QX17.3:= FALSE;
                	%QX17.5:= FALSE;
                	%QX17.4:= TRUE;
                	%QX17.6:= FALSE;
                	%QX17.7:= FALSE;
                END_IF
            }
    Group (735,42 266x428)
        Textfield (0,371 266x57), "Machine System"
            OnMouseClick:  Assign=Machine_system_properties, Type=Assignment
            OnMouseClick: execute {
                IF %QX19.1 := TRUE THEN
                	%QX19.0 := FALSE;
                	%QX19.1 := TRUE;
                	%QX19.2 := FALSE;
                	%QX19.3 := FALSE;
                	%QX19.4 := FALSE;
                	%QX19.5 := FALSE;
                	%QX18.3 := FALSE;
                END_IF
            }
        Textfield (0,0 266x57), "Hydraulic System"
            OnMouseClick:  Assign=Hydraulic_System, Type=Assignment
            OnMouseClick: execute {
                IF %QX19.5 := TRUE THEN
                	%QX19.0 := FALSE;
                	%QX19.1 := FALSE;
                	%QX19.2 := FALSE;
                	%QX19.3 := FALSE;
                	%QX19.4 := FALSE;
                	%QX19.5 := TRUE;
                	%QX18.3 := FALSE;
                END_IF
            }
        Textfield (0,92 266x57), "Cooling System"
            OnMouseClick:  Assign=Cooling_system, Type=Assignment
            OnMouseClick: execute {
                IF %QX19.4 := TRUE THEN
                	%QX19.0 := FALSE;
                	%QX19.1 := FALSE;
                	%QX19.2 := FALSE;
                	%QX19.3 := FALSE;
                	%QX19.4 := TRUE;
                	%QX19.5 := FALSE;
                	%QX18.3 := FALSE;
                END_IF
            }
        Textfield (0,184 266x57), "Simulation"
            OnMouseClick:  Assign=Control_System_Simulation, Type=Assignment
            OnMouseClick: execute {
                IF %QX19.3 := TRUE THEN
                	%QX19.0 := FALSE;
                	%QX19.1 := FALSE;
                	%QX19.2 := FALSE;
                	%QX19.3 := TRUE;
                	%QX19.4 := FALSE;
                	%QX19.5 := FALSE;
                	%QX18.3 := FALSE;
                END_IF
            }
        Textfield (0,276 266x57), "Camera System"
            OnMouseClick:  Assign=camera_system, Type=Assignment
            OnMouseClick: execute {
                IF %QX19.2 := TRUE THEN
                	%QX19.0 := FALSE;
                	%QX19.1 := FALSE;
                	%QX19.2 := TRUE;
                	%QX19.3 := FALSE;
                	%QX19.4 := FALSE;
                	%QX19.5 := FALSE;
                	%QX18.3 := FALSE;
                END_IF
            }
    Clock (803,583 162x157)
        p1016715431: Element-Clock-Green
    Label (255,-80 520x220), "WELCOME ON BOARD"
    Image (295,429 433x313), image: ImagePool.Picture1
    hotkey  Id=481043677184, Key=KeyDown=True, KeyName=KEY3_2, VisuElemId=79
    hotkey  Id=481044725760, Key=KeyName=KEY3_2, VisuElemId=79
    hotkey  Id=481045774336, Key=KeyDown=True, KeyName=KEY1_4, VisuElemId=77
    hotkey  Id=481046822912, Key=KeyName=KEY1_4, VisuElemId=77
    hotkey  Id=481047871488, Key=KeyDown=True, KeyName=KEY1_2, VisuElemId=73
    hotkey  Id=481048920064, Key=KeyName=KEY1_2, VisuElemId=73
    hotkey  Id=481049968640, Key=KeyDown=True, KeyName=KEY1_1, VisuElemId=71
    hotkey  Id=481051017216, Key=KeyName=KEY1_1, VisuElemId=71
    hotkey  Id=481052065792, Key=KeyDown=True, KeyName=KEY1_3, VisuElemId=75
    hotkey  Id=481053114368, Key=KeyName=KEY1_3, VisuElemId=75
    hotkey  Id=481054162944, Key=KeyDown=True, KeyName=KEY1_5, VisuElemId=81
    hotkey  Id=481055211520, Key=KeyName=KEY1_5, VisuElemId=81
    hotkey  Id=481056260096, Key=KeyDown=True, KeyName=KEY3_6, VisuElemId=86
    hotkey  Id=481057308672, Key=KeyName=KEY3_6, VisuElemId=86
    hotkey  Id=481058357248, Key=KeyDown=True, KeyName=KEY3_5, VisuElemId=87
    hotkey  Id=481059405824, Key=KeyName=KEY3_5, VisuElemId=87
    hotkey  Id=481060454400, Key=KeyDown=True, KeyName=KEY3_4, VisuElemId=88
    hotkey  Id=481061502976, Key=KeyName=KEY3_4, VisuElemId=88
    hotkey  Id=481062551552, Key=KeyDown=True, KeyName=KEY3_3, VisuElemId=93
    hotkey  Id=481063600128, Key=KeyName=KEY3_3, VisuElemId=93
END_VISUALIZATION

// Device/Application/Battery_sys
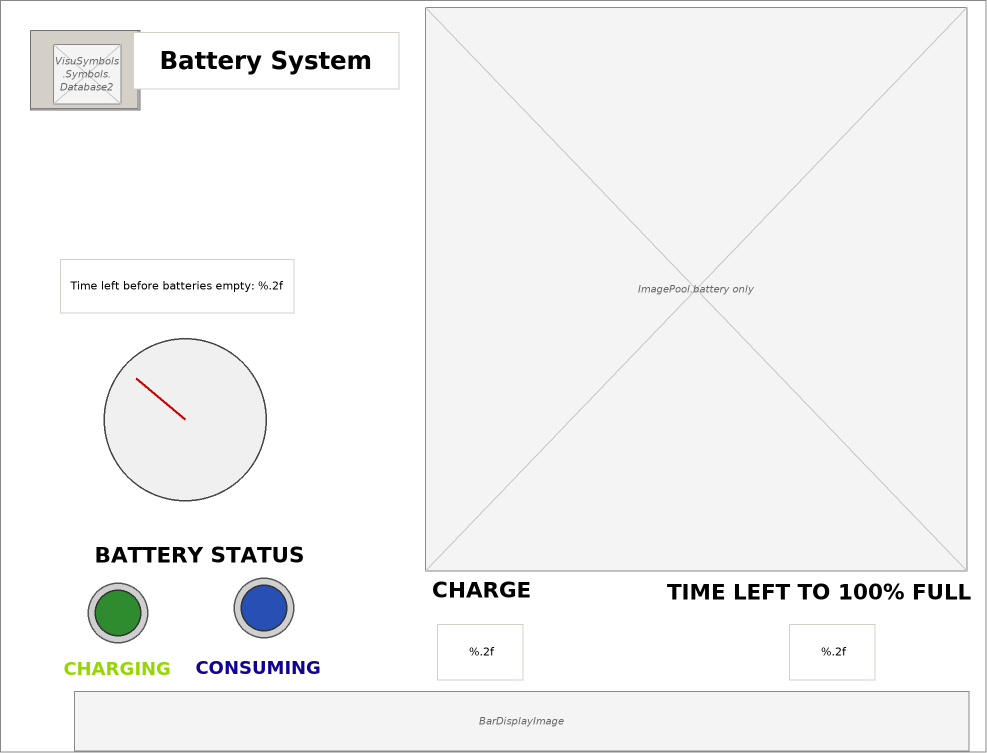
VISUALIZATION Battery_sys  // 987x753
    Group (30,30 90x60)
        OnMouseClick:  Assign=Main_sys, Type=Assignment
        OnMouseClick: execute {
            IF %QX17.0 := TRUE THEN
            	%QX17.1 := FALSE;
            	%QX17.0 := FALSE;
            END_IF
        }
        Button (0,0 110x80)
            OnMouseUp:  Assign=Main_sys, Type=Assignment
        Image (23,14 68x60), image: VisuSymbols.Symbols.Database2
            OnMouseDown:  Assign=Main_sys, Type=Assignment
    BarDisplayImage (74,691 895x60), value: PLC_PRG.tank4, style: BarDisplayImage-Gray, scale format: %.1f, scale 0..100
        p518627256: %
    Textfield (133,32 266x57), "Battery System"
        OnMouseClick:  Assign=Battery_sys, Type=Assignment
    Group (47,259 282x434)
        Meter360 (54,79 168x163), value: PLC_PRG.rate4, style: Meter-Meter360-Gray, scale format: %.1f, scale 0..100
        Label (32,272 241x48), "BATTERY STATUS"
        Textfield (13,0 234x54), "Time left before batteries empty: %.2f"
        Lamp1 (36,319 70x70), variable: PLC_PRG.charge4, style: Lamp-Lamp1-Green
        Label (0,386 141x48), "CHARGING"
        Lamp1 (182,314 70x70), variable: PLC_PRG.charge4, style: Lamp-Lamp1-Blue
        Label (141,385 141x48), "CONSUMING"
    Label (653,568 332x48), "TIME LEFT TO 100% FULL"
    Label (361,566 241x48), "CHARGE"
    Textfield (437,624 86x56), "%.2f"
    Textfield (789,624 86x56), "%.2f"
    Image (425,7 542x564), image: ImagePool.battery only
    hotkey  Id=481037385728, Key=KeyDown=True, KeyName=KEY1_1, VisuElemId=77
    hotkey  Id=481038434304, Key=KeyName=KEY1_1, VisuElemId=77
    hotkey  Id=481047871488, Key=KeyDown=True, KeyName=KEY1_2, VisuElemId=80
    hotkey  Id=481048920064, Key=KeyName=KEY1_2, VisuElemId=80
END_VISUALIZATION

// Device/Application/Hydrogen_Fuel_cell_sys
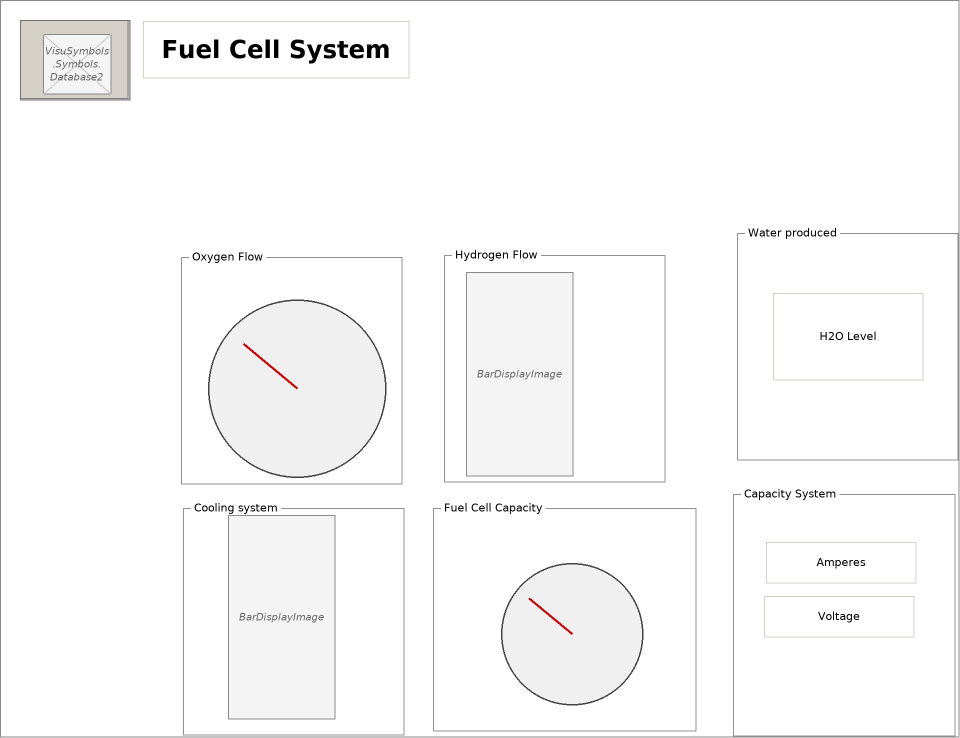
VISUALIZATION Hydrogen_Fuel_cell_sys  // 960x738
    Group (20,20 90x60)
        OnMouseClick:  Assign=Main_sys, Type=Assignment
        OnMouseClick: execute {
            IF %QX17.0 := TRUE THEN
            	%QX17.2 := FALSE;
            	%QX17.0 := FALSE;
            END_IF
        }
        Button (0,0 110x80)
            OnMouseUp:  Assign=Main_sys, Type=Assignment
        Image (23,14 68x60), image: VisuSymbols.Symbols.Database2
            OnMouseDown:  Assign=Main_sys, Type=Assignment
    GroupBox (181,249 221x235), "Oxygen Flow"
        Meter360 (27,45 178x189), style: Meter-Meter360-Gray, scale format: %.1f, scale 0..100
    GroupBox (737,225 221x235), "Water produced"
        Textfield (36,68 150x87), "H2O Level"
    GroupBox (444,247 221x235), "Hydrogen Flow"
        BarDisplayImage (22,25 107x204), style: BarDisplayImage-Gray, scale format: %.1f, scale 0..100
    GroupBox (183,500 221x235), "Cooling system"
        BarDisplayImage (45,15 107x204), style: BarDisplayImage-Gray, scale format: %.1f, scale 0..100
    GroupBox (433,500 263x231), "Fuel Cell Capacity"
        Meter180 (23,63 232x142), value: PLC_PRG.tank3, style: Meter-Meter180-Gray, scale format: %.1f, scale 0..120
    GroupBox (733,486 222x250), "Capacity System"
        Textfield (31,110 150x41), "Voltage"
        Textfield (33,56 150x41), "Amperes"
    Textfield (143,21 266x57), "Fuel Cell System"
        OnMouseClick:  Assign=Hydrogen_Fuel_cell_sys, Type=Assignment
    hotkey  Id=481037385728, Key=KeyDown=True, KeyName=KEY1_1, VisuElemId=109
    hotkey  Id=481038434304, Key=KeyName=KEY1_1, VisuElemId=109
    hotkey  Id=481052065792, Key=KeyDown=True, KeyName=KEY1_3, VisuElemId=111
    hotkey  Id=481053114368, Key=KeyName=KEY1_3, VisuElemId=111
END_VISUALIZATION

// Device/Application/Main_Overview
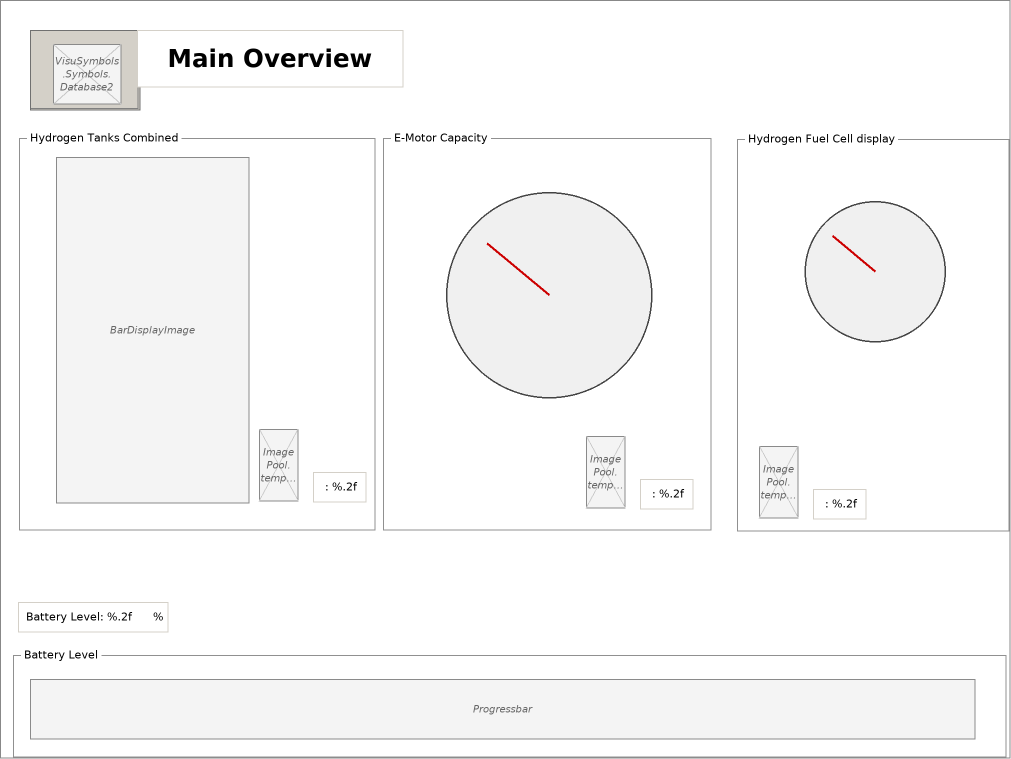
VISUALIZATION Main_Overview  // 1011x759, background image 
    GroupBox (19,130 356x400), "Hydrogen Tanks Combined"
        Group (240,299 107x73), text variable: PLC_PRG.vrate1
            Textfield (54,43 53x30), ": %.2f", text variable: PLC_PRG.rate4
            Image (0,0 39x72), image: ImagePool.temperature_icons
        BarDisplayImage (37,27 193x346), value: PLC_PRG.tank1, style: BarDisplayImage-Gray, scale format: %.1f, scale 0..100
            p518627256: Litres
    GroupBox (383,130 328x400), "E-Motor Capacity"
        Group (203,306 107x73)
            Textfield (54,43 53x30), ": %.2f", text variable: PLC_PRG.rate4
            Image (0,0 39x72), image: ImagePool.temperature_icons
        Meter360 (63,56 206x218), value: PLC_PRG.tank2, style: Meter-Meter360-Gray, scale format: %.1f, scale 0..160
    GroupBox (13,647 993x110), "Battery Level"
        Progressbar (17,32 945x60), variable: PLC_PRG.tank4
    GroupBox (737,131 272x400), "Hydrogen Fuel Cell display"
        Group (22,315 107x73)
            Textfield (54,43 53x30), ": %.2f", text variable: PLC_PRG.rate4
            Image (0,0 39x72), image: ImagePool.temperature_icons
    Meter180 (747,201 256x141), value: PLC_PRG.tank3, style: Meter-Meter180-Gray, scale format: %.1f, scale 0..120
    Group (30,30 90x60)
        OnMouseClick:  Assign=Main_sys, Type=Assignment
        OnMouseClick: execute {
            %QX17.0 := TRUE;
            	%QW8 :=	0;
            	%QX17.0:= FALSE;
        }
        OnMouseLeave:  Assign=Main_sys, Type=Assignment
        Button (0,0 110x80)
        Image (23,14 68x60), image: VisuSymbols.Symbols.Database2
            OnMouseDown:  Assign=Main_sys, Type=Assignment
    Textfield (18,602 150x30), "Battery Level: %.2f %", text variable: PLC_PRG.tank4
    Textfield (137,30 266x57), "Main Overview"
        OnMouseClick:  Assign=Main_Overview, Type=Assignment
    hotkey  Id=481037385728, Key=KeyDown=True, KeyName=KEY1_1, VisuElemId=41
    hotkey  Id=481038434304, Key=KeyName=KEY1_1, VisuElemId=41
    hotkey  Id=481049968640, Key=KeyDown=True, KeyName=KEY1_1, VisuElemId=47
    hotkey  Id=481051017216, Key=KeyName=KEY1_1, VisuElemId=47
END_VISUALIZATION

// Device/Application/Hydrogen_Tanks
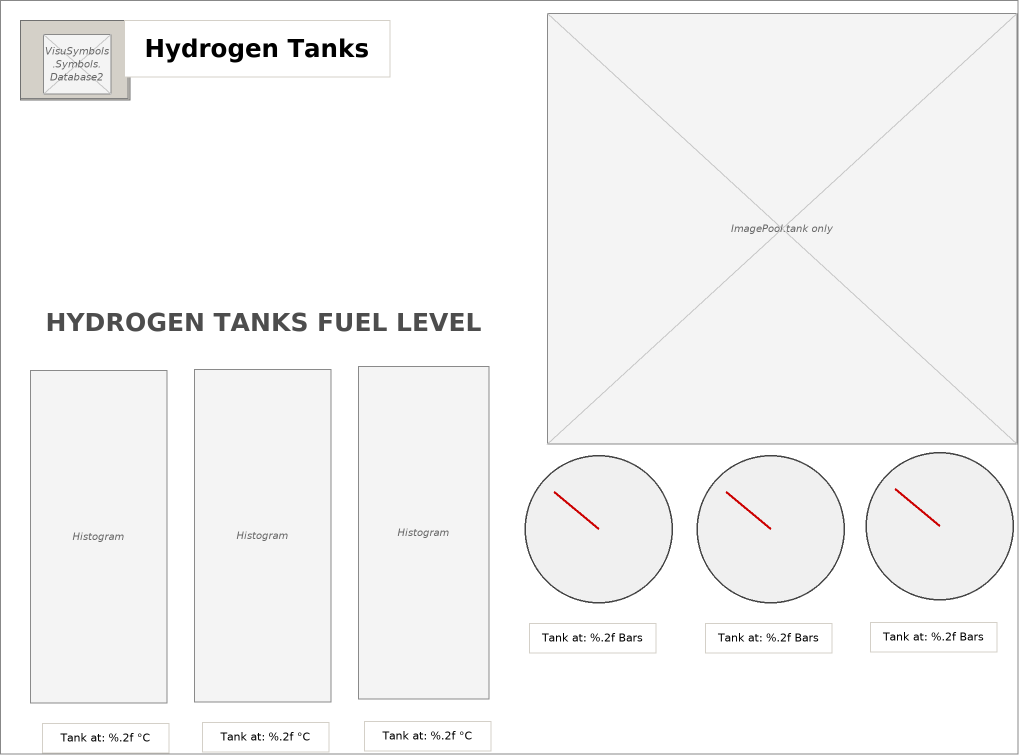
VISUALIZATION Hydrogen_Tanks  // 1019x755
    Group (20,20 90x60)
        OnMouseClick:  Assign=Main_sys, Type=Assignment
        OnMouseClick: execute {
            IF %QX17.0 := TRUE THEN
            	%QX17.4 := FALSE;
            	%QX17.0 := FALSE;
            END_IF
        }
        Button (0,0 110x80)
            OnMouseClick:  Assign=Main_sys, Type=Assignment
            OnMouseUp:  Assign=Main_sys, Type=Assignment
        Image (23,14 68x60), image: VisuSymbols.Symbols.Database2
            OnMouseClick:  Assign=Main_sys, Type=Assignment
    Histogram (30,370 137x333), scale format: %.1f, scale 0..100
        p1518820177: PLC_PRG.tank1
        p102497268: PLC_PRG.tank1
    Histogram (194,369 137x333), scale format: %.1f, scale 0..100
        p1518820177: PLC_PRG.tank1
        p102497268: PLC_PRG.tank1
    Histogram (358,366 131x333), scale format: %.1f, scale 0..100
        p1518820177: PLC_PRG.tank1
        p102497268: PLC_PRG.tank1
    Textfield (42,723 127x30), "Tank at: %.2f °C", text variable: PLC_PRG.tank1
    Textfield (124,20 266x57), "Hydrogen Tanks"
        OnMouseClick:  Assign=Hydrogen_Tanks, Type=Assignment
    Image (547,13 470x431), image: ImagePool.tank only
    Meter360 (523,455 151x148), value: PLC_PRG.tank1, style: Meter-Meter360-Gray, scale format: %.1f, scale 0..100
    Meter360 (695,455 151x148), value: PLC_PRG.tank1, style: Meter-Meter360-Gray, scale format: %.1f, scale 0..100
    Meter360 (864,452 151x148), value: PLC_PRG.tank1, style: Meter-Meter360-Gray, scale format: %.1f, scale 0..100
    Textfield (529,623 127x30), "Tank at: %.2f Bars", text variable: PLC_PRG.tank1
    Textfield (705,623 127x30), "Tank at: %.2f Bars", text variable: PLC_PRG.tank1
    Textfield (870,622 127x30), "Tank at: %.2f Bars", text variable: PLC_PRG.tank1
    Textfield (202,722 127x30), "Tank at: %.2f °C", text variable: PLC_PRG.tank1
    Textfield (364,721 127x30), "Tank at: %.2f °C", text variable: PLC_PRG.tank1
    Label (14,283 499x78), "HYDROGEN TANKS FUEL LEVEL"
    hotkey  Id=481037385728, Key=KeyDown=True, KeyName=KEY1_1, VisuElemId=49
    hotkey  Id=481038434304, Key=KeyName=KEY1_1, VisuElemId=49
    hotkey  Id=481054162944, Key=KeyDown=True, KeyName=KEY1_6, VisuElemId=59
    hotkey  Id=481055211520, Key=KeyName=KEY1_6, VisuElemId=59
END_VISUALIZATION

// Device/Application/Machine_system_properties
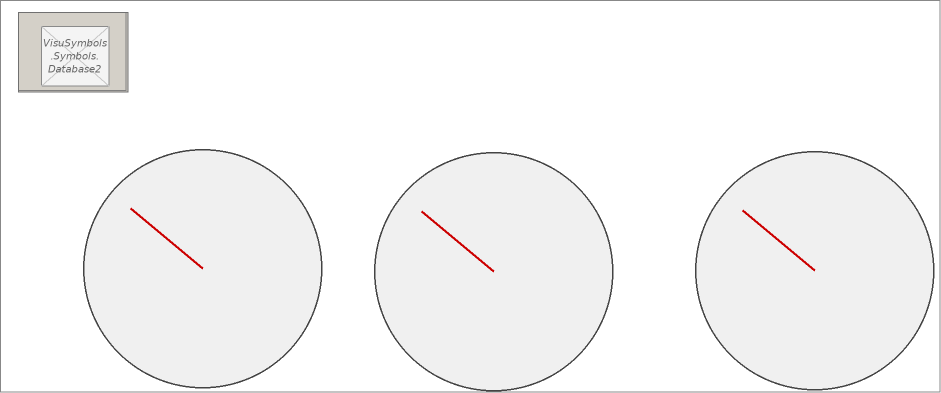
VISUALIZATION Machine_system_properties  // 941x393
    Group (18,12 110x80)
        OnMouseClick:  Assign=Main_sys, Type=Assignment
        OnMouseClick: execute {
            IF %QX17.0 := TRUE THEN
            	%QX19.1 := FALSE;
            	%QX17.0 := FALSE;
            END_IF
        }
        Button (0,0 110x80)
            OnMouseUp:  Assign=Main_sys, Type=Assignment
        Image (23,14 68x60), image: VisuSymbols.Symbols.Database2
            OnMouseClick:  Assign=Main_sys, Type=Assignment
    Meter360 (78,149 249x239), value: PLC_PRG.longi, style: Meter-Meter360-Gray, scale format: %.1f, scale 0..4000
    Meter360 (369,152 249x239), value: PLC_PRG.slope, style: Meter-Meter360-Gray, scale format: %.1f, scale 0..4000
    Meter360 (690,151 249x239), value: PLC_PRG.x_vector1, style: Meter-Meter360-Gray, scale format: %.1f, scale 0..4000
    hotkey  Id=481037385728, Key=KeyDown=True, KeyName=KEY1_1, VisuElemId=5
    hotkey  Id=481038434304, Key=KeyName=KEY1_1, VisuElemId=5
END_VISUALIZATION

// Device/Application/Control_System_Simulation
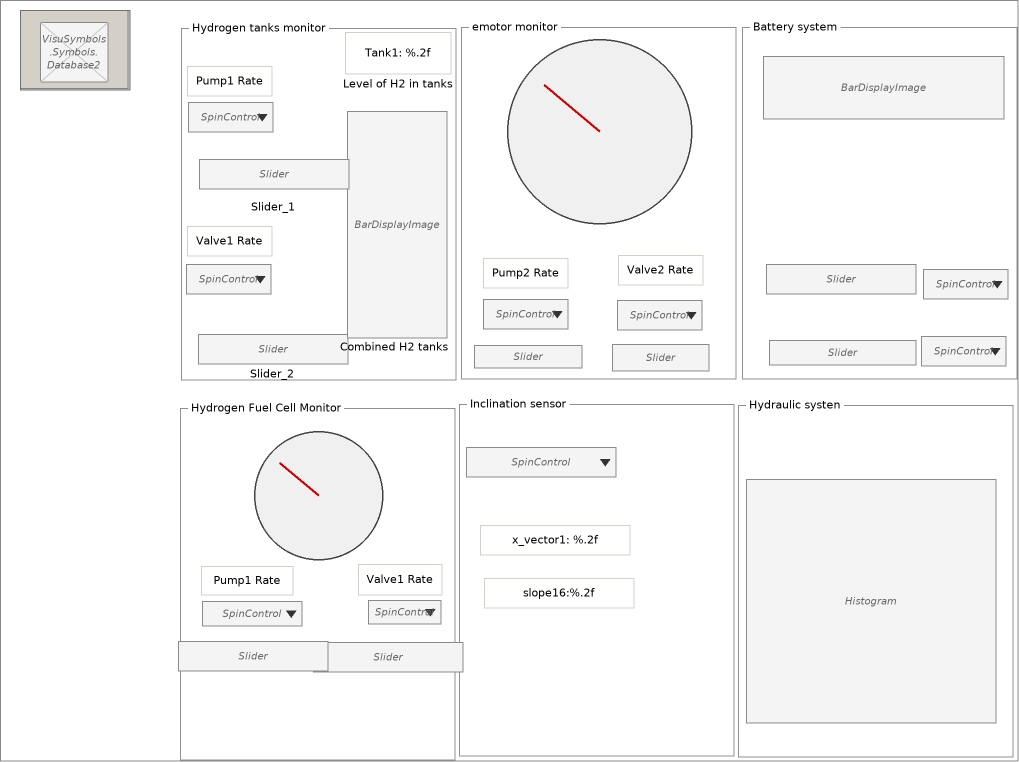
VISUALIZATION Control_System_Simulation  // 1019x762
    GroupBox (181,20 275x360), "Hydrogen tanks monitor"
        Slider (17,314 150x30), variable: PLC_PRG.vrate1, scale 0..100
        BarDisplayImage (166,91 100x227), value: PLC_PRG.tank1, style: BarDisplayImage-Gray, scale format: %.1f, scale 0..100
        SpinControl (5,244 85x30), variable: PLC_PRG.vrate1
        Textfield (6,206 85x30), "Valve1 Rate"
        SpinControl (7,82 85x30), variable: PLC_PRG.rate1
        Textfield (6,46 85x30), "Pump1 Rate"
        Textfield (164,12 106x42), "Tank1: %.2f", text variable: PLC_PRG.tank1
        Slider (18,139 150x30), variable: PLC_PRG.rate1, scale 0..100
        Label (17,172 150x30), "Slider_1"
    GroupBox (461,19 275x360), "emotor monitor"
        Meter360 (38,20 201x185), value: PLC_PRG.tank2, style: Meter-Meter360-Gray, scale format: %.1f, scale 0..160
        Textfield (157,236 85x30), "Valve2 Rate"
        SpinControl (156,281 85x30), variable: PLC_PRG.vrate2
        Slider (151,325 97x27), variable: PLC_PRG.vrate2, scale 0..100
        Textfield (22,239 85x30), "Pump2 Rate"
        SpinControl (22,280 85x30), variable: PLC_PRG.rate2
        Slider (13,326 108x23), variable: PLC_PRG.rate2, scale 0..100
    GroupBox (742,19 275x360), "Battery system"
        Slider (24,245 150x30), variable: PLC_PRG.rate4, scale 0..100
        Slider (27,321 147x25), variable: PLC_PRG.vrate4, scale 0..100
        SpinControl (181,250 85x30), variable: PLC_PRG.rate4
        SpinControl (179,317 85x30), variable: PLC_PRG.vrate4
        BarDisplayImage (21,37 241x63), value: PLC_PRG.tank4, style: BarDisplayImage-Gray, scale format: %.1f, scale 0..100
            p518627256: %
    GroupBox (180,400 275x360), "Hydrogen Fuel Cell Monitor"
        Meter180 (29,31 219x129), value: PLC_PRG.tank3, style: Meter-Meter180-Gray, scale format: %.1f, scale 0..120
        Textfield (21,166 92x29), "Pump1 Rate"
        SpinControl (22,201 100x25), variable: PLC_PRG.rate3
        Textfield (178,164 84x31), "Valve1 Rate"
        SpinControl (188,200 73x24), variable: PLC_PRG.vrate3
    GroupBox (459,396 275x360), "Inclination sensor"
        SpinControl (7,51 150x30), variable: PLC_PRG.x_vector1
            p576042468: -100
        Textfield (21,129 150x30), "x_vector1: %.2f", text variable: PLC_PRG.x_vector1
        Textfield (25,182 150x30), "slope16:%.2f", text variable: PLC_PRG.slope
    GroupBox (738,397 275x360), "Hydraulic systen"
        Histogram (8,82 250x244), scale format: %.1f, scale 0..100
            p1518820177: PLC_PRG.tank2
            p102497268: PLC_PRG.tank2
    Group (20,10 90x60)
        OnMouseClick:  Assign=Main_sys, Type=Assignment
        OnMouseClick: execute {
            IF %QX17.0 := TRUE THEN
            	%QW9 := 0;
            	%QX17.0 := FALSE;
            END_IF
        }
        Button (0,0 110x80)
            OnMouseClick:  Assign=Main_sys, Type=Assignment
            OnMouseDown:  Assign=Main_sys, Type=Assignment
        Image (20,12 68x60), image: VisuSymbols.Symbols.Database2
            OnMouseDown:  Assign=Main_sys, Type=Assignment
    Slider (313,642 150x30), variable: PLC_PRG.vrate3, scale 0..100
    Slider (178,641 150x30), variable: PLC_PRG.rate3, scale 0..100
    Label (197,359 150x30), "Slider_2"
    Label (319,332 150x30), "Combined H2 tanks"
    Label (323,69 150x30), "Level of H2 in tanks"
    hotkey  Id=481037385728, Key=KeyDown=True, KeyName=KEY1_1, VisuElemId=33
    hotkey  Id=481038434304, Key=KeyName=KEY1_1, VisuElemId=33
    hotkey  Id=481039482880, Key=KeyDown=True, KeyName=KEY1_1, VisuElemId=104
    hotkey  Id=481040531456, Key=KeyName=KEY1_1, VisuElemId=104
END_VISUALIZATION

// Device/Application/Visualization
VISUALIZATION Visualization  // 2x2
END_VISUALIZATION

// Device/Application/electric_motor
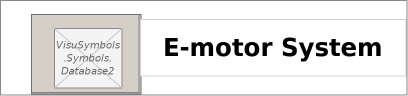
VISUALIZATION electric_motor  // 408x96
    Group (31,14 90x60)
        OnMouseClick:  Assign=Main_sys, Type=Assignment
        OnMouseClick: execute {
            IF %QX17.0 := TRUE THEN
            	%QX17.3 := FALSE;
            	%QX17.0 := FALSE;
            END_IF
        }
        Button (0,0 110x80)
            OnMouseUp:  Assign=Main_sys, Type=Assignment
        Image (23,14 68x60), image: VisuSymbols.Symbols.Database2
            OnMouseDown:  Assign=Main_sys, Type=Assignment
    Textfield (140,19 266x57), "E-motor System"
    hotkey  Id=481037385728, Key=KeyDown=True, KeyName=KEY1_1, VisuElemId=3
    hotkey  Id=481038434304, Key=KeyName=KEY1_1, VisuElemId=3
    hotkey  Id=481045774336, Key=KeyDown=True, KeyName=KEY1_4, VisuElemId=5
    hotkey  Id=481046822912, Key=KeyName=KEY1_4, VisuElemId=5
END_VISUALIZATION

// Device/Application/Hydraulic_System
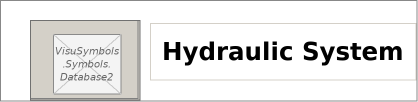
VISUALIZATION Hydraulic_System  // 418x102
    Group (30,20 90x60)
        OnMouseClick:  Assign=Main_sys, Type=Assignment
        OnMouseClick: execute {
            IF %QX17.0 := TRUE THEN
            	%QX17.0 := FALSE;
            	%QX19.5 := FALSE;
            END_IF
        }
        Button (0,0 110x80)
            OnMouseUp:  Assign=Main_sys, Type=Assignment
        Image (23,14 68x60), image: VisuSymbols.Symbols.Database2
            OnMouseDown:  Assign=Main_sys, Type=Assignment
    Textfield (150,23 266x57), "Hydraulic System"
        OnMouseClick:  Assign=Hydraulic_System, Type=Assignment
    hotkey  Id=481037385728, Key=KeyDown=True, KeyName=KEY1_1, VisuElemId=3
    hotkey  Id=481038434304, Key=KeyName=KEY1_1, VisuElemId=3
END_VISUALIZATION

// Device/Application/Cooling_system
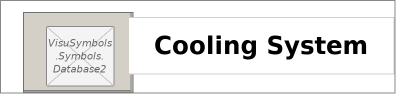
VISUALIZATION Cooling_system  // 396x94
    Group (23,12 90x60)
        OnMouseClick:  Assign=Main_sys, Type=Assignment
        OnMouseClick: execute {
            IF %QX17.0 := TRUE THEN
            	%QX19.4 := FALSE;
            	%QX17.0 := FALSE;
            END_IF
        }
        Button (0,0 110x80)
            OnMouseUp:  Assign=Main_sys, Type=Assignment
        Image (23,14 68x60), image: VisuSymbols.Symbols.Database2
            OnMouseDown:  Assign=Main_sys, Type=Assignment
    Textfield (128,17 266x57), "Cooling System"
        OnMouseClick:  Assign=Hydrogen_Fuel_cell_sys, Type=Assignment
    hotkey  Id=481037385728, Key=KeyDown=True, KeyName=KEY1_1, VisuElemId=3
    hotkey  Id=481038434304, Key=KeyName=KEY1_1, VisuElemId=3
END_VISUALIZATION

// Device/Application/camera_system
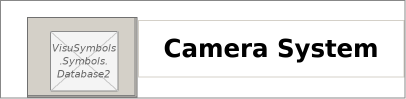
VISUALIZATION camera_system  // 406x99
    Group (27,17 90x60)
        OnMouseClick:  Assign=Main_sys, Type=Assignment
        OnMouseClick: execute {
            IF %QX17.0 := TRUE THEN
            	%QX19.2 := FALSE;
            	%QX17.0 := FALSE;
            END_IF
        }
        Button (0,0 110x80)
            OnMouseUp:  Assign=Main_sys, Type=Assignment
        Image (23,14 68x60), image: VisuSymbols.Symbols.Database2
            OnMouseDown:  Assign=Main_sys, Type=Assignment
    Textfield (138,20 266x57), "Camera System"
    hotkey  Id=481037385728, Key=KeyDown=True, KeyName=KEY1_1, VisuElemId=3
    hotkey  Id=481038434304, Key=KeyName=KEY1_1, VisuElemId=3
END_VISUALIZATION

(* text list System (id | default)
  Apr | Apr
  April | April
  Aug | Aug
  August | August
  Dec | Dec
  December | December
  Feb | Feb
  February | February
  Fri | Fri
  Friday | Friday
  Jan | Jan
  January | January
  Jul | Jul
  July | July
  Jun | Jun
  June | June
  Mar | Mar
  March | March
  May | May
  May_3Letter | May
  Mon | Mon
  Monday | Monday
  Nov | Nov
  November | November
  Oct | Oct
  October | October
  Sat | Sat
  Saturday | Saturday
  Sep | Sep
  September | September
  Sun | Sun
  Sunday | Sunday
  Thu | Thu
  Thursday | Thursday
  Tue | Tue
  Tuesday | Tuesday
  Wed | Wed
  Wednesday | Wednesday
   |  *)
